FUNCTION_BLOCK LfcPrint
  (* Standard: 61499-2 *)
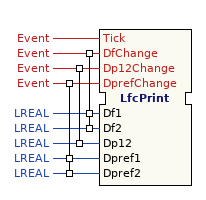
  EVENT_INPUT
    Tick;
    DfChange WITH Df1, Df2;
    Dp12Change WITH Dp12;
    DprefChange WITH Dpref1, Dpref2;
  END_EVENT
  VAR_INPUT
    Df1 : LREAL;
    Df2 : LREAL;
    Dp12 : LREAL;
    Dpref1 : LREAL;
    Dpref2 : LREAL;
  END_VAR
END_FUNCTION_BLOCK
(* other elements stored in the file *)
(* Autogenerate Language=C ArbitraryText= #include <stdio.h> #include <stdlib.h> RunText= if(me->inputEvents.event.Tick) { static int tickCount = 0; static int firstRun = 1; if(firstRun == 1) { printf("%10s, %10s, %10s, %10s, %10s, %10s\r\n", "Time", "Dpref1", "Dpref2", "Df1", "Df2", "Dp12"); firstRun = 0; } printf("%10f, %10f, %10f, %10f, %10f, %10f\r\n", tickCount * 0.1, me->Dpref1, me->Dpref2, me->Df1, me->Df2, me->Dp12); tickCount++; } me->inputEvents.event.Tick = 0; *)
